Fanuc KAREL source: kb00106.KL

-- PROVISIONAL review KL for V940-1; original PC SHA256 e96d7b45721106022a39a74bebf4a83b81691f815839f08680a555cda9dca584
-- Incomplete behavior may be omitted. Consult companion uncertainty JSON. Do not deploy.
PROGRAM KB00106
%NOLOCKGROUP
BEGIN
  -- V9_ZERO_TABLE_METADATA_HINT layout=0002_ascii; no indexed target words; source/name/runtime held
  -- UNRESOLVED_PC offsets 5-15; opcodes 27,22,31
  -- UNRESOLVED_PC offsets 20-24; opcodes 7F
END KB00106
